INTERFACE ITF_MCHMIPrepareScreen_01_XX_Init

METHOD PUBLIC LinkDataHMI_01_XX : BOOL
VAR_INPUT
	refstData				: REFERENCE TO ST_MCHMIPrepareScreen_01_XX;
END_VAR
END_METHOD

END_INTERFACE

(* stored: Version 1.1.0.1
   Itf ITF_MCHMIPrepareScreen_01_XX_Init: Id {bd2ed89e-f866-0789-3b0b-6f16927b846b}
   Method LinkDataHMI_01_XX: Id {d37b8c5f-6239-0f40-3a0b-235fd0502426} *)
